FUNCTION_BLOCK FB_LoadingModeChange
VAR_INPUT
	LoadingModeSelected : eLoadingMode;	
	LS_AutoMode		: BOOL;
	LS_ManualMode	: BOOL;
	LS_SemiAutoMode : BOOL; 
END_VAR
VAR_OUTPUT
	PS_AutoMode		: BOOL;
	PS_ManualMode	: BOOL;
	PS_SemiAutoMode : BOOL;
END_VAR
VAR_IN_OUT
	ActualMode : eLoadingMode;
END_VAR
VAR
	RTRIG_AutoMode :  R_TRIG;
	RTRIG_ManualMode :  R_TRIG;
	RTRIG_SemiAutoMode :  R_TRIG;
END_VAR

RTRIG_AutoMode(CLK := LS_AutoMode);
RTRIG_ManualMode(CLK := LS_ManualMode);
RTRIG_SemiAutoMode(CLK := LS_SemiAutoMode);

//IF LoadingModeSelected <> ActualMode THEN
	IF LoadingModeSelected = eLoadingMOde.Auto THEN
		PS_AutoMode := TRUE;
		PS_ManualMode := FALSE;
		PS_SemiAutoMOde := FALSE;
	ELSIF LoadingModeSelected = eLoadingMOde.Manual THEN
		PS_AutoMode := FALSE;
		PS_ManualMode := TRUE;
		PS_SemiAutoMOde := FALSE;
	ELSIF LoadingModeSelected = eLoadingMOde.SemiAuto THEN
		PS_AutoMode := FALSE;
		PS_ManualMode := FALSE;
		PS_SemiAutoMOde := TRUE;
	ELSE
		PS_AutoMode := FALSE;
		PS_ManualMode := FALSE;
		PS_SemiAutoMOde := FALSE;		
	END_IF
//END_IF

IF RTRIG_AutoMode.Q THEN
	PS_AutoMode := FALSE;
	PS_ManualMode := FALSE;
	PS_SemiAutoMOde := FALSE;
	ActualMode := eLoadingMode.Auto;	
END_IF

IF RTRIG_ManualMode.Q THEN
	PS_AutoMode := FALSE;
	PS_ManualMode := FALSE;
	PS_SemiAutoMOde := FALSE;
	ActualMode := eLoadingMode.Manual;	
END_IF

IF RTRIG_SemiAutoMode.Q THEN
	PS_AutoMode := FALSE;
	PS_ManualMode := FALSE;
	PS_SemiAutoMOde := FALSE;
	ActualMode := eLoadingMode.SemiAuto;	
END_IF

END_FUNCTION_BLOCK

(* stored: Version 1.1.0.1, ProductVersion 3.1.4024.15
   POU FB_LoadingModeChange: Id {bdf76c89-1c98-4edb-9f2e-18c9b359c7a1}, SpecialFunc None *)
